INTERFACE I_AlarmVisitor

METHOD VisitAlarm
VAR_INPUT
	VisitingAlarm : I_Alarm;
END_VAR
END_METHOD

END_INTERFACE

(* stored: Version 1.1.0.1, ProductVersion 3.1.4024.12
   Itf I_AlarmVisitor: Id {66b3db5f-9868-4317-b709-8cea6ef4ca14}
   Method VisitAlarm: Id {24923fb7-4c34-47be-9e63-4b0b306988aa} *)
